Staubli VAL3: txt_PkgInit.pgx

program txt_PkgInit()
begin
  call TxtReadRoom1()
  if nTxtTotal>1
    call TxtReadRoom2()
  endIf
end
